                         IF #password <> #EMPTY_WSTRING AND #username <> #EMPTY_WSTRING
                         THEN
                           #tempPasswordFlag := TRUE;
                           FOR #tempLoopCounter := #FIRST_CHARACTER TO LEN(#password) DO
                             "LMQTT_ConvertToUtf8"(character     := #password[#tempLoopCounter],
                                                   convertedUtf8 => #tempConvertedUtf8,
                                                   bytesUsed     => #tempBytesUsedUtf8,
                                                   error         => #tempErrorConvertUtf8,
                                                   status        => #tempStatusConvertUtf8);
                             #statPasswordLenUtf8Encoded := #statPasswordLenUtf8Encoded + #tempBytesUsedUtf8;
                           END_FOR;
                           #statSendPaketTotalRemLen := #statSendPaketTotalRemLen + #statPasswordLenUtf8Encoded + #TWO_BYTE_LEN_INFO;
                         ELSE
                           #statPasswordEncodeState := #NOT_USED_NO_ENCODING;
                           #tempPasswordFlag := FALSE;
                         END_IF;


                         IF #willtopic <> #EMPTY_WSTRING
                         THEN
                           #tempWillFlag := TRUE;
                           CASE #statWillQos OF
                             #MQTT_QOS_0:  // Statement section case 1
                               #tempWillQoS1 := FALSE;
                               #tempWillQoS2 := FALSE;
                             #MQTT_QOS_1:  // Statement section case 2 to 4
                               #tempWillQoS1 := TRUE;
                               #tempWillQoS2 := FALSE;
                             #MQTT_QOS_2:
                               #tempWillQoS1 := FALSE;
                               #tempWillQoS2 := True;
                             ELSE  // Statement section ELSE
                               ;
                           END_CASE;
                           FOR #tempLoopCounter := #FIRST_CHARACTER TO LEN(#willtopic) DO
                             // Statement section FOR
                             "LMQTT_ConvertToUtf8"(character     := #willtopic[#tempLoopCounter],
                                                   convertedUtf8 => #tempConvertedUtf8,
                                                   bytesUsed     => #tempBytesUsedUtf8,
                                                   error         => #tempErrorConvertUtf8,
                                                   status        => #tempStatusConvertUtf8);
                             #statWillTopicLenUtf8Encoded := #statWillTopicLenUtf8Encoded + #tempBytesUsedUtf8;
                           END_FOR;
                           //Add WillTopic Len and Will Message Len (and len info twice)
                           #statSendPaketTotalRemLen := #statSendPaketTotalRemLen + #statWillTopicLenUtf8Encoded + #statWillMessageCnt + (2 * #TWO_BYTE_LEN_INFO);
                         ELSE
                           #statWillTopicEncodeState := #NOT_USED_NO_ENCODING;
                           #statWillMessageEncodeState := #NOT_USED_NO_ENCODING;
                           #tempWillFlag := FALSE;
                           #statWillRetain := FALSE;
                           #tempWillQoS1 := FALSE;
                           #tempWillQoS2 := FALSE;
                         END_IF;

                         //Build Connect Telegram
                         //Fixed Header - Write Paket Type
                         #statSendBuffer[#statSendBufferPos] := #MQTT_MSG_TYPE_CONNECT; // 1 Byte
                         #statSendBufferPos += 1; // increment

                         //Write Remaining Paket Len info 
                         WHILE (#statSendPaketTotalRemLen > #DEFAULT_VALUE_ZERO)
                         DO//See MQTT Spec for explanation of this calculation
                           #statEncodedRemPaketLenAsByte := UDINT_TO_BYTE(#statSendPaketTotalRemLen MOD #SEND_LEN_MULTIPLIER_UDINT_128);
                           #statSendPaketTotalRemLen := #statSendPaketTotalRemLen / #SEND_LEN_MULTIPLIER_UDINT_128;
                           // if there are more data to encode, set the top bit of this byte
                           IF #statSendPaketTotalRemLen > #DEFAULT_VALUE_ZERO
                           THEN
                             // Do this and continue while loop
                             #statEncodedRemPaketLenAsByte := #statEncodedRemPaketLenAsByte OR UDINT_TO_BYTE(#SEND_LEN_MULTIPLIER_UDINT_128);
                             #statSendBuffer[#statSendBufferPos] := #statEncodedRemPaketLenAsByte;
                             #statSendBufferPos += 1;
                           ELSE
                             //do this and leave while loop
                             #statSendBuffer[#statSendBufferPos] := #statEncodedRemPaketLenAsByte;
                             #statSendBufferPos += 1;
                           END_IF;
                         END_WHILE;

                         //Build Connect Telegram
                         // Write Protocol name
                         #statSendBuffer[#statSendBufferPos] := #CONN_PROTOCOL_NAME_0;
                         #statSendBufferPos += 1;
                         #statSendBuffer[#statSendBufferPos] := #CONN_PROTOCOL_NAME_4;
                         #statSendBufferPos += 1;
                         #statSendBuffer[#statSendBufferPos] := CHAR_TO_BYTE('M');
                         #statSendBufferPos += 1;
                         #statSendBuffer[#statSendBufferPos] := CHAR_TO_BYTE('Q');
                         #statSendBufferPos += 1;
                         #statSendBuffer[#statSendBufferPos] := CHAR_TO_BYTE('T');
                         #statSendBufferPos += 1;
                         #statSendBuffer[#statSendBufferPos] := CHAR_TO_BYTE('T');
                         #statSendBufferPos += 1;
                         //Write Protocol Level
                         #statSendBuffer[#statSendBufferPos] := #CONN_PROTOCOL_MQTT_VERSION_3_1_1;
                         #statSendBufferPos += 1;
                         //Write Connect Flags
                         #statSendBuffer[#statSendBufferPos].%X0 := false;
                         #statSendBuffer[#statSendBufferPos].%X1 := True;
                         #statSendBuffer[#statSendBufferPos].%X2 := #tempWillFlag;
                         #statSendBuffer[#statSendBufferPos].%X3 := #tempWillQoS1;
                         #statSendBuffer[#statSendBufferPos].%X4 := #tempWillQoS2;
                         #statSendBuffer[#statSendBufferPos].%X5 := #statWillRetain;
                         #statSendBuffer[#statSendBufferPos].%X6 := #tempPasswordFlag;
                         #statSendBuffer[#statSendBufferPos].%X7 := #tempUserFlag;
                         #statSendBufferPos += 1;
                         //Write Keep Alive in sec
                         #tempWordForSliceAddress := UINT_TO_WORD(#connParam.keepAlive);
                         #statSendBuffer[#statSendBufferPos] := #tempWordForSliceAddress.%B1;
                         #statSendBufferPos += 1;
                         #statSendBuffer[#statSendBufferPos] := #tempWordForSliceAddress.%B0;
                         #statSendBufferPos += 1;

                         //Set To Complete this, can skip in further progess
                         #statPaketHeaderEncodeDone := TRUE;
                       END_IF;

                       // Payload
                       // These fields, if present, MUST appear in the order:
                       // Client Identifier, Will topic, Will message, User Name, password


                       //ClientIdentifier
                       IF #statSendBufferPos <= #MAX_BUFFER_LEN_SEND - #TWO_BYTE_LEN_INFO THEN
                         CASE #statClientIdEncodeState OF
                           #FIRST_ENCODING:  // Statement section case 1
                             //ADD len info into paket

                             #tempWordForSliceAddress := UINT_TO_WORD(#statClientIdLenUtf8Encoded);
                             #statSendBuffer[#statSendBufferPos] := #tempWordForSliceAddress.%B1; //MSB
                             #statSendBufferPos += 1;
                             #statSendBuffer[#statSendBufferPos] := #tempWordForSliceAddress.%B0; // LSB
                             #statSendBufferPos += 1;

                             FOR #tempLoopCounter := #statClientIdPos TO LEN(#clientIdentifier) DO
                               "LMQTT_ConvertToUtf8"(character     := #clientIdentifier[#tempLoopCounter],
                                                     convertedUtf8 => #tempConvertedUtf8,
                                                     bytesUsed     => #tempBytesUsedUtf8,
                                                     error         => #tempErrorConvertUtf8,
                                                     status        => #tempStatusConvertUtf8);

                               IF #statSendBufferPos + #tempBytesUsedUtf8 <= #MAX_BUFFER_LEN_SEND THEN
                                 #statClientIdPos += 1;
                                 CASE #tempBytesUsedUtf8 OF
                                   #UTF_1_BYTE_USED:  // Statement section case 1
                                     #statSendBuffer[#statSendBufferPos] := #tempConvertedUtf8.%B0;
                                     #statSendBufferPos += 1;
                                   #UTF_2_BYTE_USED:
                                     #statSendBuffer[#statSendBufferPos] := #tempConvertedUtf8.%B0;
                                     #statSendBufferPos += 1;
                                     #statSendBuffer[#statSendBufferPos] := #tempConvertedUtf8.%B1;
                                     #statSendBufferPos += 1;
                                   #UTF_3_BYTE_USED:  // Statement section case 2 to 4
                                     #statSendBuffer[#statSendBufferPos] := #tempConvertedUtf8.%B0;
                                     #statSendBufferPos += 1;
                                     #statSendBuffer[#statSendBufferPos] := #tempConvertedUtf8.%B1;
                                     #statSendBufferPos += 1;
                                     #statSendBuffer[#statSendBufferPos] := #tempConvertedUtf8.%B2;
                                     #statSendBufferPos += 1;
                                   ELSE  // Statement section ELSE
                                     ;
                                 END_CASE;
                               ELSE
                                 //When buffer full
                                 #statClientIdEncodeState := #SUBSEQUENT_ENCODING;
                                 EXIT;
                               END_IF;
                             END_FOR;
                             IF #statClientIdPos >= LEN(#clientIdentifier) THEN
                               #statClientIdEncodeState := #ENCODE_DONE;
                             END_IF;


                           #SUBSEQUENT_ENCODING:  // Statement section case 2 to 4
                             FOR #tempLoopCounter := #statClientIdPos TO LEN(#clientIdentifier) DO
                               "LMQTT_ConvertToUtf8"(character     := #clientIdentifier[#tempLoopCounter],
                                                     convertedUtf8 => #tempConvertedUtf8,
                                                     bytesUsed     => #tempBytesUsedUtf8,
                                                     error         => #tempErrorConvertUtf8,
                                                     status        => #tempStatusConvertUtf8);
                               IF #statSendBufferPos + #tempBytesUsedUtf8 <= #MAX_BUFFER_LEN_SEND THEN
                                 #statClientIdPos += 1;
                                 CASE #tempBytesUsedUtf8 OF
                                   #UTF_1_BYTE_USED:  // Statement section case 1
                                     #statSendBuffer[#statSendBufferPos] := #tempConvertedUtf8.%B0;
                                     #statSendBufferPos += 1;
                                   #UTF_2_BYTE_USED:
                                     #statSendBuffer[#statSendBufferPos] := #tempConvertedUtf8.%B0;
                                     #statSendBufferPos += 1;
                                     #statSendBuffer[#statSendBufferPos] := #tempConvertedUtf8.%B1;
                                     #statSendBufferPos += 1;
                                   #UTF_3_BYTE_USED:  // Statement section case 2 to 4
                                     #statSendBuffer[#statSendBufferPos] := #tempConvertedUtf8.%B0;
                                     #statSendBufferPos += 1;
                                     #statSendBuffer[#statSendBufferPos] := #tempConvertedUtf8.%B1;
                                     #statSendBufferPos += 1;
                                     #statSendBuffer[#statSendBufferPos] := #tempConvertedUtf8.%B2;
                                     #statSendBufferPos += 1;
                                   ELSE  // Statement section ELSE
                                     ;
                                 END_CASE;
                               ELSE
                                 //When buffer full
                                 EXIT;
                               END_IF;
                             END_FOR;
                             IF #statClientIdPos >= LEN(#clientIdentifier) THEN
                               #statClientIdEncodeState := #ENCODE_DONE;
                             END_IF;
                           ELSE  // Statement section ELSE
                             ; // IDLE / SKIP
                         END_CASE;
                       END_IF;

                       // Will Topic
                       // If the Will Flag is set to 1, the Will Topic is the next field in the payload. It must be > 0 Bytes

                       IF #statClientIdEncodeState = #ENCODE_DONE
                         AND #statSendBufferPos <= #MAX_BUFFER_LEN_SEND - #TWO_BYTE_LEN_INFO THEN
                         //When Client Id is encoded and buffer not full
                         //And willTopic is used
                         CASE #statWillTopicEncodeState OF
                           #FIRST_ENCODING:  // Statement section case 1
                             //ADD len info into paket

                             #tempWordForSliceAddress := UINT_TO_WORD(#statWillTopicLenUtf8Encoded);
                             #statSendBuffer[#statSendBufferPos] := #tempWordForSliceAddress.%B1; //MSB
                             #statSendBufferPos += 1;
                             #statSendBuffer[#statSendBufferPos] := #tempWordForSliceAddress.%B0; // LSB
                             #statSendBufferPos += 1;

                             FOR #tempLoopCounter := #statWillTopicPos TO LEN(#willtopic) DO
                               "LMQTT_ConvertToUtf8"(character     := #willtopic[#tempLoopCounter],
                                                     convertedUtf8 => #tempConvertedUtf8,
                                                     bytesUsed     => #tempBytesUsedUtf8,
                                                     error         => #tempErrorConvertUtf8,
                                                     status        => #tempStatusConvertUtf8);

                               IF #statSendBufferPos + #tempBytesUsedUtf8 <= #MAX_BUFFER_LEN_SEND THEN
                                 //Increment when successful
                                 #statWillTopicPos += 1;

                                 CASE #tempBytesUsedUtf8 OF
                                   #UTF_1_BYTE_USED:  // Statement section case 1
                                     #statSendBuffer[#statSendBufferPos] := #tempConvertedUtf8.%B0;
                                     #statSendBufferPos += 1;
                                   #UTF_2_BYTE_USED:
                                     #statSendBuffer[#statSendBufferPos] := #tempConvertedUtf8.%B0;
                                     #statSendBufferPos += 1;
                                     #statSendBuffer[#statSendBufferPos] := #tempConvertedUtf8.%B1;
                                     #statSendBufferPos += 1;
                                   #UTF_3_BYTE_USED:  // Statement section case 2 to 4
                                     #statSendBuffer[#statSendBufferPos] := #tempConvertedUtf8.%B0;
                                     #statSendBufferPos += 1;
                                     #statSendBuffer[#statSendBufferPos] := #tempConvertedUtf8.%B1;
                                     #statSendBufferPos += 1;
                                     #statSendBuffer[#statSendBufferPos] := #tempConvertedUtf8.%B2;
                                     #statSendBufferPos += 1;
                                   ELSE  // Statement section ELSE
                                     ;
                                 END_CASE;
                               ELSE
                                 //When buffer full
                                 #statWillTopicEncodeState := #SUBSEQUENT_ENCODING;
                                 EXIT;
                               END_IF;
                             END_FOR;

                             IF #statWillTopicPos >= LEN(#willtopic) THEN
                               #statWillTopicEncodeState := #ENCODE_DONE;
                             END_IF;

                           #SUBSEQUENT_ENCODING:  // Statement section case 2 to 4
                             FOR #tempLoopCounter := #statWillTopicPos TO LEN(#willtopic) DO
                               "LMQTT_ConvertToUtf8"(character     := #willtopic[#tempLoopCounter],
                                                     convertedUtf8 => #tempConvertedUtf8,
                                                     bytesUsed     => #tempBytesUsedUtf8,
                                                     error         => #tempErrorConvertUtf8,
                                                     status        => #tempStatusConvertUtf8);

                               IF #statSendBufferPos + #tempBytesUsedUtf8 <= #MAX_BUFFER_LEN_SEND THEN
                                 #statWillTopicPos += 1;
                                 CASE #tempBytesUsedUtf8 OF
                                   #UTF_1_BYTE_USED:  // Statement section case 1
                                     #statSendBuffer[#statSendBufferPos] := #tempConvertedUtf8.%B0;
                                     #statSendBufferPos += 1;
                                   #UTF_2_BYTE_USED:
                                     #statSendBuffer[#statSendBufferPos] := #tempConvertedUtf8.%B0;
                                     #statSendBufferPos += 1;
                                     #statSendBuffer[#statSendBufferPos] := #tempConvertedUtf8.%B1;
                                     #statSendBufferPos += 1;
                                   #UTF_3_BYTE_USED:  // Statement section case 2 to 4
                                     #statSendBuffer[#statSendBufferPos] := #tempConvertedUtf8.%B0;
                                     #statSendBufferPos += 1;
                                     #statSendBuffer[#statSendBufferPos] := #tempConvertedUtf8.%B1;
                                     #statSendBufferPos += 1;
                                     #statSendBuffer[#statSendBufferPos] := #tempConvertedUtf8.%B2;
                                     #statSendBufferPos += 1;
                                   ELSE  // Statement section ELSE
                                     ;
                                 END_CASE;
                               ELSE
                                 //When buffer full
                                 EXIT;
                               END_IF;
                             END_FOR;
                             IF #statWillTopicPos >= LEN(#willtopic) THEN
                               #statWillTopicEncodeState := #ENCODE_DONE;
                             END_IF;

                           ELSE  // Statement section ELSE
                             ;
                         END_CASE;
                       END_IF;

                       // Will Message
                       // This field consists OF a two Byte length followed BY the payload FOR the Will message expressed as a sequence bytes.

                       IF #statClientIdEncodeState = #ENCODE_DONE
                         AND #statWillTopicEncodeState = #ENCODE_DONE
                         AND #statSendBufferPos <= #MAX_BUFFER_LEN_SEND - #TWO_BYTE_LEN_INFO THEN
                         //When Client Id is encoded and buffer not full
                         CASE #statWillMessageEncodeState OF
                           #FIRST_ENCODING:  // Statement section case 1
                             //ADD len info into paket

                             #tempWordForSliceAddress := UINT_TO_WORD(#statWillMessageCnt);
                             #statSendBuffer[#statSendBufferPos] := #tempWordForSliceAddress.%B1; //MSB
                             #statSendBufferPos += 1;
                             #statSendBuffer[#statSendBufferPos] := #tempWordForSliceAddress.%B0; // LSB
                             #statSendBufferPos += 1;

                             #tempLowerWillMsgArrayBoundary := LOWER_BOUND(ARR := #willMsgPayload, DIM := #ONE_DIMENSION);

                             FOR #tempLoopCounter := #statWillMessagePos TO UINT_TO_DINT(#statWillMessageCnt - 1) DO
                               IF #statSendBufferPos <= #MAX_BUFFER_LEN_SEND THEN
                                 #statSendBuffer[#statSendBufferPos] := #willMsgPayload[#tempLowerWillMsgArrayBoundary + #tempLoopCounter];
                                 #statSendBufferPos += 1;
                                 //Increment when successful
                                 #statWillMessagePos += 1;
                               ELSE
                                 //When buffer full
                                 #statWillMessageEncodeState := #SUBSEQUENT_ENCODING;
                                 EXIT;
                               END_IF;
                             END_FOR;
                             // If everything was copied successfull
                             IF #statWillMessagePos >= #statWillMessageCnt THEN
                               #statWillMessageEncodeState := #ENCODE_DONE;
                             END_IF;

                           #SUBSEQUENT_ENCODING:  // Statement section case 2 to 4
                             #tempLowerWillMsgArrayBoundary := LOWER_BOUND(ARR := #willMsgPayload, DIM := #ONE_DIMENSION);

                             FOR #tempLoopCounter := #statWillMessagePos TO UINT_TO_DINT(#statWillMessageCnt - 1) DO
                               IF #statSendBufferPos <= #MAX_BUFFER_LEN_SEND THEN
                                 #statSendBuffer[#statSendBufferPos] := #willMsgPayload[#tempLowerWillMsgArrayBoundary + #tempLoopCounter];
                                 #statSendBufferPos += 1;
                                 //Increment when successful
                                 #statWillMessagePos += 1;
                               ELSE
                                 //When Buffer Full
                                 EXIT;
                               END_IF;
                             END_FOR;
                             // If everything was copied successfull
                             IF #statWillMessagePos >= #statWillMessageCnt THEN
                               #statWillMessageEncodeState := #ENCODE_DONE;
                             END_IF;


                           ELSE  // Statement section ELSE
                             ;
                         END_CASE;
                       END_IF;

                       // Username
                       // If the Username Flag is set to 1, the Username the next field in the payload. It must be > 0 Bytes

                       IF #statClientIdEncodeState = #ENCODE_DONE
                         AND (#statWillTopicEncodeState = #ENCODE_DONE OR #statWillTopicEncodeState = #NOT_USED_NO_ENCODING)
                         AND (#statWillMessageEncodeState = #ENCODE_DONE OR #statWillTopicEncodeState = #NOT_USED_NO_ENCODING)
                         AND #statSendBufferPos <= #MAX_BUFFER_LEN_SEND - #TWO_BYTE_LEN_INFO THEN
                         //When Will Topic and Will Message is encoded and buffer not full
                         CASE #statUserNameEncodeState OF
                           #FIRST_ENCODING:  // Statement section case 1
                             //ADD len info into paket

                             #tempWordForSliceAddress := UINT_TO_WORD(#statUsernameLenUtf8Encoded);
                             #statSendBuffer[#statSendBufferPos] := #tempWordForSliceAddress.%B1; //MSB
                             #statSendBufferPos += 1;
                             #statSendBuffer[#statSendBufferPos] := #tempWordForSliceAddress.%B0; // LSB
                             #statSendBufferPos += 1;

                             FOR #tempLoopCounter := #statUserNamePos TO LEN(#username) DO
                               "LMQTT_ConvertToUtf8"(character     := #username[#tempLoopCounter],
                                                     convertedUtf8 => #tempConvertedUtf8,
                                                     bytesUsed     => #tempBytesUsedUtf8,
                                                     error         => #tempErrorConvertUtf8,
                                                     status        => #tempStatusConvertUtf8);

                               IF #statSendBufferPos + #tempBytesUsedUtf8 <= #MAX_BUFFER_LEN_SEND THEN
                                 //Increment when successful
                                 #statUserNamePos += 1;

                                 CASE #tempBytesUsedUtf8 OF
                                   #UTF_1_BYTE_USED:  // Statement section case 1
                                     #statSendBuffer[#statSendBufferPos] := #tempConvertedUtf8.%B0;
                                     #statSendBufferPos += 1;
                                   #UTF_2_BYTE_USED:
                                     #statSendBuffer[#statSendBufferPos] := #tempConvertedUtf8.%B0;
                                     #statSendBufferPos += 1;
                                     #statSendBuffer[#statSendBufferPos] := #tempConvertedUtf8.%B1;
                                     #statSendBufferPos += 1;
                                   #UTF_3_BYTE_USED:  // Statement section case 2 to 4
                                     #statSendBuffer[#statSendBufferPos] := #tempConvertedUtf8.%B0;
                                     #statSendBufferPos += 1;
                                     #statSendBuffer[#statSendBufferPos] := #tempConvertedUtf8.%B1;
                                     #statSendBufferPos += 1;
                                     #statSendBuffer[#statSendBufferPos] := #tempConvertedUtf8.%B2;
                                     #statSendBufferPos += 1;
                                   ELSE  // Statement section ELSE
                                     ;
                                 END_CASE;
                               ELSE
                                 //When buffer full
                                 #statUserNameEncodeState := #SUBSEQUENT_ENCODING;
                                 EXIT;
                               END_IF;
                             END_FOR;

                             IF #statUserNamePos >= LEN(#username) THEN
                               #statUserNameEncodeState := #ENCODE_DONE;
                             END_IF;

                           #SUBSEQUENT_ENCODING:  // Statement section case 2 to 4
                             FOR #tempLoopCounter := #statUserNamePos TO LEN(#username) DO
                               "LMQTT_ConvertToUtf8"(character     := #username[#tempLoopCounter],
                                                     convertedUtf8 => #tempConvertedUtf8,
                                                     bytesUsed     => #tempBytesUsedUtf8,
                                                     error         => #tempErrorConvertUtf8,
                                                     status        => #tempStatusConvertUtf8);

                               IF #statSendBufferPos + #tempBytesUsedUtf8 <= #MAX_BUFFER_LEN_SEND THEN
                                 #statUserNamePos += 1;
                                 CASE #tempBytesUsedUtf8 OF
                                   #UTF_1_BYTE_USED:  // Statement section case 1
                                     #statSendBuffer[#statSendBufferPos] := #tempConvertedUtf8.%B0;
                                     #statSendBufferPos += 1;
                                   #UTF_2_BYTE_USED:
                                     #statSendBuffer[#statSendBufferPos] := #tempConvertedUtf8.%B0;
                                     #statSendBufferPos += 1;
                                     #statSendBuffer[#statSendBufferPos] := #tempConvertedUtf8.%B1;
                                     #statSendBufferPos += 1;
                                   #UTF_3_BYTE_USED:  // Statement section case 2 to 4
                                     #statSendBuffer[#statSendBufferPos] := #tempConvertedUtf8.%B0;
                                     #statSendBufferPos += 1;
                                     #statSendBuffer[#statSendBufferPos] := #tempConvertedUtf8.%B1;
                                     #statSendBufferPos += 1;
                                     #statSendBuffer[#statSendBufferPos] := #tempConvertedUtf8.%B2;
                                     #statSendBufferPos += 1;
                                   ELSE  // Statement section ELSE
                                     ;
                                 END_CASE;
                               ELSE
                                 //When buffer full
                                 EXIT;
                               END_IF;
                             END_FOR;
                             IF #statUserNamePos >= LEN(#username) THEN
                               #statUserNameEncodeState := #ENCODE_DONE;
                             END_IF;

                           ELSE  // Statement section ELSE
                             ;
                         END_CASE;
                       END_IF;

                       // Password
                       // If the Password Flag is set to 1, the Password the next field in the payload. It must be > 0 Bytes
                       //Password field contains 0 to 65535 bytes OF binary data prefixed with a two Byte length field which indicates the number OF bytes used

                       IF #statClientIdEncodeState = #ENCODE_DONE
                         AND (#statWillTopicEncodeState = #ENCODE_DONE OR #statWillTopicEncodeState = #NOT_USED_NO_ENCODING)
                         AND (#statWillMessageEncodeState = #ENCODE_DONE OR #statWillMessageEncodeState = #NOT_USED_NO_ENCODING)
                         AND (#statUserNameEncodeState = #ENCODE_DONE OR #statUserNameEncodeState = #NOT_USED_NO_ENCODING)
                         AND #statSendBufferPos <= #MAX_BUFFER_LEN_SEND - #TWO_BYTE_LEN_INFO THEN
                         //When Will Topic and Will Message is encoded and buffer not full
                         CASE #statPasswordEncodeState OF
                           #FIRST_ENCODING:  // Statement section case 1
                             //ADD len info into paket

                             #tempWordForSliceAddress := UINT_TO_WORD(#statPasswordLenUtf8Encoded);
                             #statSendBuffer[#statSendBufferPos] := #tempWordForSliceAddress.%B1; //MSB
                             #statSendBufferPos += 1;
                             #statSendBuffer[#statSendBufferPos] := #tempWordForSliceAddress.%B0; // LSB
                             #statSendBufferPos += 1;

                             FOR #tempLoopCounter := #statPasswordPos TO LEN(#password) DO
                               "LMQTT_ConvertToUtf8"(character     := #password[#tempLoopCounter],
                                                     convertedUtf8 => #tempConvertedUtf8,
                                                     bytesUsed     => #tempBytesUsedUtf8,
                                                     error         => #tempErrorConvertUtf8,
                                                     status        => #tempStatusConvertUtf8);

                               IF #statSendBufferPos + #tempBytesUsedUtf8 <= #MAX_BUFFER_LEN_SEND THEN
                                 //Increment when successful
                                 #statPasswordPos += 1;

                                 CASE #tempBytesUsedUtf8 OF
                                   #UTF_1_BYTE_USED:  // Statement section case 1
                                     #statSendBuffer[#statSendBufferPos] := #tempConvertedUtf8.%B0;
                                     #statSendBufferPos += 1;
                                   #UTF_2_BYTE_USED:
                                     #statSendBuffer[#statSendBufferPos] := #tempConvertedUtf8.%B0;
                                     #statSendBufferPos += 1;
                                     #statSendBuffer[#statSendBufferPos] := #tempConvertedUtf8.%B1;
                                     #statSendBufferPos += 1;
                                   #UTF_3_BYTE_USED:  // Statement section case 2 to 4
                                     #statSendBuffer[#statSendBufferPos] := #tempConvertedUtf8.%B0;
                                     #statSendBufferPos += 1;
                                     #statSendBuffer[#statSendBufferPos] := #tempConvertedUtf8.%B1;
                                     #statSendBufferPos += 1;
                                     #statSendBuffer[#statSendBufferPos] := #tempConvertedUtf8.%B2;
                                     #statSendBufferPos += 1;
                                   ELSE  // Statement section ELSE
                                     ;
                                 END_CASE;
                               ELSE
                                 //When buffer full
                                 #statPasswordEncodeState := #SUBSEQUENT_ENCODING;
                                 EXIT;
                               END_IF;
                             END_FOR;

                             IF #statPasswordPos >= LEN(#password) THEN
                               #statPasswordEncodeState := #ENCODE_DONE;
                             END_IF;

                           #SUBSEQUENT_ENCODING:  // Statement section case 2 to 4
                             FOR #tempLoopCounter := #statPasswordPos TO LEN(#password) DO
                               "LMQTT_ConvertToUtf8"(character     := #password[#tempLoopCounter],
                                                     convertedUtf8 => #tempConvertedUtf8,
                                                     bytesUsed     => #tempBytesUsedUtf8,
                                                     error         => #tempErrorConvertUtf8,
                                                     status        => #tempStatusConvertUtf8);

                               IF #statSendBufferPos + #tempBytesUsedUtf8 <= #MAX_BUFFER_LEN_SEND THEN
                                 #statPasswordPos += 1;
                                 CASE #tempBytesUsedUtf8 OF
                                   #UTF_1_BYTE_USED:  // Statement section case 1
                                     #statSendBuffer[#statSendBufferPos] := #tempConvertedUtf8.%B0;
                                     #statSendBufferPos += 1;
                                   #UTF_2_BYTE_USED:
                                     #statSendBuffer[#statSendBufferPos] := #tempConvertedUtf8.%B0;
                                     #statSendBufferPos += 1;
                                     #statSendBuffer[#statSendBufferPos] := #tempConvertedUtf8.%B1;
                                     #statSendBufferPos += 1;
                                   #UTF_3_BYTE_USED:  // Statement section case 2 to 4
                                     #statSendBuffer[#statSendBufferPos] := #tempConvertedUtf8.%B0;
                                     #statSendBufferPos += 1;
                                     #statSendBuffer[#statSendBufferPos] := #tempConvertedUtf8.%B1;
                                     #statSendBufferPos += 1;
                                     #statSendBuffer[#statSendBufferPos] := #tempConvertedUtf8.%B2;
                                     #statSendBufferPos += 1;
                                   ELSE  // Statement section ELSE
                                     ;
                                 END_CASE;
                               ELSE
                                 //When buffer full
                                 EXIT;
                               END_IF;
                             END_FOR;
                             IF #statPasswordPos >= LEN(#password) THEN
                               #statPasswordEncodeState := #ENCODE_DONE;
                             END_IF;

                           ELSE  // Statement section ELSE
                             ;
                         END_CASE;
                       END_IF;

                       //set Sendlen for TSendC Block

                       #statTsendcLen := #statSendBufferPos; // Buffer pos equals amount of elements in send array
                       //reset buffer pos
                       #statSendBufferPos := 0;
                       //enable Send Req
                       #statTsendcReq := TRUE;
                       //Set Watchdog
                       #statEnableTimerCommandWatchdog := TRUE;
                       //wait for send to be done
                       #statMqttConnectState := #MQTT_CONNECT_STATE_SEND_PAKET_WAIT_FOR_CONNACK;
                     END_IF;
                   END_REGION BUILD_CONNECT_PAKET
                 #MQTT_CONNECT_STATE_SEND_PAKET_WAIT_FOR_CONNACK:
                   REGION SEND_CONNECT_PAKET_WAIT_FOR_CONNACK
                     //check tsend status
                     IF NOT #tempTsendcBusy AND #tempTsendcStatus = #TSENDC_JOB_DONE THEN
                       IF (#statClientIdEncodeState = #ENCODE_DONE OR #statClientIdEncodeState = #NOT_USED_NO_ENCODING)
                         AND (#statWillTopicEncodeState = #ENCODE_DONE OR #statWillTopicEncodeState = #NOT_USED_NO_ENCODING)
                         AND (#statWillMessageEncodeState = #ENCODE_DONE OR #statWillMessageEncodeState = #NOT_USED_NO_ENCODING)
                         AND (#statUserNameEncodeState = #ENCODE_DONE OR #statUserNameEncodeState = #NOT_USED_NO_ENCODING)
                         AND (#statPasswordEncodeState = #ENCODE_DONE OR #statPasswordEncodeState = #NOT_USED_NO_ENCODING) THEN
                         //Encoding done all sent
                         #statPaketHeaderEncodeDone := FALSE;
                       ELSE
                         // More to Encode and send
                         #statEnableTimerCommandWatchdog := FALSE;
                         #statMqttConnectState := #MQTT_CONNECT_STATE_BUILD_PAKET;
                       END_IF;
                     END_IF;
                     //Check watchdog
                     IF #instTimerCommandWatchdog.Q THEN
                       #statEnableTimerCommandWatchdog := FALSE;
                       #statPaketHeaderEncodeDone := FALSE;
                       #statStatus := #ERR_MQTT_CONNECT_TIMEOUT; // Set correct status that identifies error clearly
                       #statSubfunctionStatus := #ERR_MQTT_CONNECT_TIMEOUT; // Status or return value of called FBs, FCs and system blocks
                       #statFBErrorState := #statFBState; // Set error state number for diagnostic 
                       #statErrorAutoCleared := TRUE;
                       #statMqttConnectState := #MQTT_CONNECT_STATE_BUILD_PAKET;
                     END_IF;

                     //Check Connect ACK paket
                     CASE #tempMqttConnAckRcvStatus OF
                       #NO_RESPONSE:  //  IDLE
                         ;
                       #RESPONSE_GOOD:  // Statement section case 2 to 4
                         //disable watchdog
                         #statEnableTimerCommandWatchdog := FALSE;
                         //Encoding done all sent
                         #statPaketHeaderEncodeDone := FALSE;
                         //Go to Connected
                         #statMqttConnectState := #MQTT_CONNECT_STATE_CONNECTED;
                         #statStatus := #STATUS_MQTT_CONNECTED;
                     END_CASE;
                   END_REGION REGION SEND_CONNECT_PAKET
                 #MQTT_CONNECT_STATE_CONNECTED:
                   REGION CONNECTED
                     //Check Rising edge of input commands
                     #tempCommandInput.%X0 := #tempPublish AND NOT #statPublishOld;
                     #tempCommandInput.%X1 := #tempSubscribe AND NOT #statSubscribeOld;
                     #tempCommandInput.%X2 := #tempUnsubscribe AND NOT #statUnsubscribeOld;

                     //Start the keepalive timer if used
                     #statEnableMqttKeepAliveTimer := #statMqttKeepAliveUsed;

                     //set status to connected after successfully executed job
                     IF #statStatus = #STATUS_JOB_EXECUTED THEN
                       #statStatus := #STATUS_MQTT_CONNECTED;
                     END_IF;

                     REGION MQTT_COMMANDS
                       //When state machine is ready for a new input then assign correct command
                       //Ping job can be overwritten by a command.
                         IF #tempCommandInput <> #NO_COMMAND
                         AND (#statMqttCommandState = #MQTT_COMMAND_STATE_NO_PROCESSING OR #statMqttCommandState = #MQTT_COMMAND_STATE_SEND_PING)
                       THEN
                         // New Input set, reset done flag
                         #statDone := FALSE;
                         #statMqttCommandState := BYTE_TO_DINT(#tempCommandInput);
                       END_IF;

                       CASE #statMqttCommandState OF
                         #MQTT_COMMAND_STATE_NO_PROCESSING:
                           //EMPTY STATE
                           ;
                         #MQTT_COMMAND_STATE_BUILD_PUBLISH:  // Statement section case 1
                           REGION PUBLISH_TO_TOPIC
                             //Remaining Length is the length of the variable header (TOPIC NAME + PacketID) plus the length of the Payload. 
                             //Max Len of Mqtt pakets is per Standard 268,435,455 Bytes (ff,ff,ff,7f)
                             //Calculate Remain Len will be
                             //Len of TOPIC   (max 3*16382 WChars= 49.146 Bytes)
                             //plus Len of PacketID (2 Bytes)
                             //plus Len of Payload (max 268,435,455 - 49.146 - 2 = 268.386.307 Bytes ca. 268 MB)
                             //Max Array / DB Len in TIA portal is around 16 MB or 16.777.216 Byte
                             //Set Status
                             #statStatus := #STATUS_MQTT_PUBLISH;

                             // Must obey, if not currently sending PubAck Msg on a subscription
                             // Else, try in the next cycle
                             IF #tempTsendcBusy = FALSE // when tsendC is ready
                               AND #tempTsendcDone = FALSE // tsendC did not finish in this cycle
                               AND #statTsendcReq = FALSE // TsendC request was not already requested by pub ack msg
                             THEN
                               IF #statPaketHeaderEncodeDone = FALSE THEN

                                 //Init
                                 #statSendPaketTotalRemLen := 0;
                                 #statSendBufferPos := 0;
                                 #statPublishQos := #qos;
                                 #statPublishMessageCnt := #publishMsgLen;
                                 #statPublishTopicEncodeState := #FIRST_ENCODING;
                                 #statPublishTopicPos := #FIRST_CHARACTER;
                                 #statPublishTopicLenUtf8Encoded := 0;
                                 #statPaketId += 1;//increment
                                 #statPaketIdEncoded := FALSE;
                                 #statPublishEncodeMessageState := #SUBSEQUENT_ENCODING; // No len info necessary so start directly at subsequent.
                                 #statPublishMessagePos := 0; // first array element

                                 //verify PayloadLen
                                 #tempMaxPublishDataArrayLen := ABS(UPPER_BOUND(ARR := #publishMsgPayload, DIM := #ONE_DIMENSION) - LOWER_BOUND(ARR := #publishMsgPayload, DIM := #ONE_DIMENSION)) + #ARRAY_LEN_OFFSET_PLUS_1;

                                 //check necessary boundaries
                                 IF #tempMaxPublishDataArrayLen < #statPublishMessageCnt THEN
                                   #statStatus := #ERR_CNT_EXCEEDS_ARRAY_DIMENSION; // Set correct status that identifies error clearly
                                   #statSubfunctionStatus := #ERR_CNT_EXCEEDS_ARRAY_DIMENSION; // Status or return value of called FBs, FCs and system blocks
                                   #statFBErrorState := #statFBState; // Set error state number for diagnostic 
                                   #statErrorAutoCleared := TRUE;
                                   #statMqttCommandState := #MQTT_COMMAND_STATE_NO_PROCESSING;
                                 ELSIF LEN(#mqttTopic) = #LEN_NULL THEN
                                   #statStatus := #ERR_MQTT_COMMAND_PUBLISH_TOPIC_INVALID; // Set correct status that identifies error clearly
                                   #statSubfunctionStatus := #ERR_MQTT_COMMAND_PUBLISH_TOPIC_INVALID; // Status or return value of called FBs, FCs and system blocks
                                   #statFBErrorState := #statFBState; // Set error state number for diagnostic 
                                   #statErrorAutoCleared := TRUE;
                                   #statMqttCommandState := #MQTT_COMMAND_STATE_NO_PROCESSING;
                                 ELSIF #statPublishQos > #MQTT_QOS_2 THEN
                                   #statStatus := #ERR_QOS_INVALID; // Set correct status that identifies error clearly
                                   #statSubfunctionStatus := #ERR_QOS_INVALID; // Status or return value of called FBs, FCs and system blocks
                                   #statFBErrorState := #statFBState; // Set error state number for diagnostic 
                                   #statErrorAutoCleared := TRUE;
                                   #statMqttCommandState := #MQTT_COMMAND_STATE_NO_PROCESSING;
                                 ELSE // All ok
                                   //Add amount of bytes for publish message
                                   #statSendPaketTotalRemLen := #statSendPaketTotalRemLen + #statPublishMessageCnt;
                                   //add publish  topic len
                                   FOR #tempLoopCounter := #FIRST_CHARACTER TO LEN(#mqttTopic) DO
                                     "LMQTT_ConvertToUtf8"(character     := #mqttTopic[#tempLoopCounter],
                                                           convertedUtf8 => #tempConvertedUtf8,
                                                           bytesUsed     => #tempBytesUsedUtf8,
                                                           error         => #tempErrorConvertUtf8,
                                                           status        => #tempStatusConvertUtf8);
                                     #statPublishTopicLenUtf8Encoded := #statPublishTopicLenUtf8Encoded + #tempBytesUsedUtf8;
                                   END_FOR;
                                   #statSendPaketTotalRemLen := #statSendPaketTotalRemLen + #statPublishTopicLenUtf8Encoded + #TWO_BYTE_LEN_INFO;

                                   //Build Publish Telegram
                                   //Fixed Header - Write Paket Type
                                   #statSendBuffer[#statSendBufferPos] := #MQTT_MSG_TYPE_PUBLISH;
                                   // Set DUP flag always to FALSE
                                   #statSendBuffer[#statSendBufferPos].%X3 := FALSE;
                                   // Set QoS Level
                                   CASE #statPublishQos OF
                                     #MQTT_QOS_0:  // Statement section case 0
                                       #statSendBuffer[#statSendBufferPos].%X2 := FALSE;
                                       #statSendBuffer[#statSendBufferPos].%X1 := FALSE;
                                     #MQTT_QOS_1:  // Statement section case 1
                                       #statSendBuffer[#statSendBufferPos].%X2 := FALSE;
                                       #statSendBuffer[#statSendBufferPos].%X1 := TRUE;
                                       //Add two byte len info for Mandatory packet ID
                                       #statSendPaketTotalRemLen := #statSendPaketTotalRemLen + #TWO_BYTE_LEN_INFO;
                                     #MQTT_QOS_2: // Statement section case 2
                                       #statSendBuffer[#statSendBufferPos].%X2 := TRUE;
                                       #statSendBuffer[#statSendBufferPos].%X1 := FALSE;
                                       //Add two byte len info for Mandatory packet ID
                                       #statSendPaketTotalRemLen := #statSendPaketTotalRemLen + #TWO_BYTE_LEN_INFO;
                                     ELSE
                                       ;
                                   END_CASE;
                                   //Set retain bit
                                   #statSendBuffer[#statSendBufferPos].%X0 := #retain;

                                   #statSendBufferPos += 1; // increment

                                   //Write Remaining Paket Len info 
                                   WHILE (#statSendPaketTotalRemLen > #DEFAULT_VALUE_ZERO)
                                   DO//See MQTT Spec for explanation of this calculation
                                     #statEncodedRemPaketLenAsByte := UDINT_TO_BYTE(#statSendPaketTotalRemLen MOD #SEND_LEN_MULTIPLIER_UDINT_128);
                                     #statSendPaketTotalRemLen := #statSendPaketTotalRemLen / #SEND_LEN_MULTIPLIER_UDINT_128;
                                     // if there are more data to encode, set the top bit of this byte
                                     IF #statSendPaketTotalRemLen > #DEFAULT_VALUE_ZERO
                                     THEN
                                       // Do this and continue while loop
                                       #statEncodedRemPaketLenAsByte := #statEncodedRemPaketLenAsByte OR UDINT_TO_BYTE(#SEND_LEN_MULTIPLIER_UDINT_128);
                                       #statSendBuffer[#statSendBufferPos] := #statEncodedRemPaketLenAsByte;
                                       #statSendBufferPos += 1;
                                     ELSE
                                       //do this and leave while loop
                                       #statSendBuffer[#statSendBufferPos] := #statEncodedRemPaketLenAsByte;
                                       #statSendBufferPos += 1;
                                     END_IF;
                                   END_WHILE;
                                   //When all done, set encode to true
                                   #statPaketHeaderEncodeDone := TRUE;
                                 END_IF;
                               END_IF;

                               //Header Encoded - now Topic, PacketId and Message need to be encoded.
                               IF #statPaketHeaderEncodeDone = TRUE THEN

                                 //Publish Topic
                                 IF #statSendBufferPos <= #MAX_BUFFER_LEN_SEND - #TWO_BYTE_LEN_INFO THEN
                                   CASE #statPublishTopicEncodeState OF
                                     #FIRST_ENCODING:  // Statement section case 1
                                       //ADD len info into paket

                                       #tempWordForSliceAddress := UINT_TO_WORD(#statPublishTopicLenUtf8Encoded);
                                       #statSendBuffer[#statSendBufferPos] := #tempWordForSliceAddress.%B1; //MSB
                                       #statSendBufferPos += 1;
                                       #statSendBuffer[#statSendBufferPos] := #tempWordForSliceAddress.%B0; // LSB
                                       #statSendBufferPos += 1;

                                       FOR #tempLoopCounter := #statPublishTopicPos TO LEN(#mqttTopic) DO
                                         "LMQTT_ConvertToUtf8"(character     := #mqttTopic[#tempLoopCounter],
                                                               convertedUtf8 => #tempConvertedUtf8,
                                                               bytesUsed     => #tempBytesUsedUtf8,
                                                               error         => #tempErrorConvertUtf8,
                                                               status        => #tempStatusConvertUtf8);

                                         IF #statSendBufferPos + #tempBytesUsedUtf8 <= #MAX_BUFFER_LEN_SEND THEN
                                           #statPublishTopicPos += 1;
                                           CASE #tempBytesUsedUtf8 OF
                                             #UTF_1_BYTE_USED:  // Statement section case 1
                                               #statSendBuffer[#statSendBufferPos] := #tempConvertedUtf8.%B0;
                                               #statSendBufferPos += 1;
                                             #UTF_2_BYTE_USED:
                                               #statSendBuffer[#statSendBufferPos] := #tempConvertedUtf8.%B0;
                                               #statSendBufferPos += 1;
                                               #statSendBuffer[#statSendBufferPos] := #tempConvertedUtf8.%B1;
                                               #statSendBufferPos += 1;
                                             #UTF_3_BYTE_USED:  // Statement section case 2 to 4
                                               #statSendBuffer[#statSendBufferPos] := #tempConvertedUtf8.%B0;
                                               #statSendBufferPos += 1;
                                               #statSendBuffer[#statSendBufferPos] := #tempConvertedUtf8.%B1;
                                               #statSendBufferPos += 1;
                                               #statSendBuffer[#statSendBufferPos] := #tempConvertedUtf8.%B2;
                                               #statSendBufferPos += 1;
                                             ELSE  // Statement section ELSE
                                               ;
                                           END_CASE;
                                         ELSE
                                           //When buffer full
                                           #statPublishTopicEncodeState := #SUBSEQUENT_ENCODING;
                                           EXIT;
                                         END_IF;
                                       END_FOR;
                                       IF #statPublishTopicPos >= LEN(#mqttTopic) THEN
                                         #statPublishTopicEncodeState := #ENCODE_DONE;
                                       END_IF;


                                     #SUBSEQUENT_ENCODING:  // Statement section case 2 to 4
                                       FOR #tempLoopCounter := #statPublishTopicPos TO LEN(#mqttTopic) DO

                                         "LMQTT_ConvertToUtf8"(character     := #mqttTopic[#tempLoopCounter],
                                                               convertedUtf8 => #tempConvertedUtf8,
                                                               bytesUsed     => #tempBytesUsedUtf8,
                                                               error         => #tempErrorConvertUtf8,
                                                               status        => #tempStatusConvertUtf8);
                                         IF #statSendBufferPos + #tempBytesUsedUtf8 <= #MAX_BUFFER_LEN_SEND THEN
                                           #statPublishTopicPos += 1;
                                           CASE #tempBytesUsedUtf8 OF
                                             #UTF_1_BYTE_USED:  // Statement section case 1
                                               #statSendBuffer[#statSendBufferPos] := #tempConvertedUtf8.%B0;
                                               #statSendBufferPos += 1;
                                             #UTF_2_BYTE_USED:
                                               #statSendBuffer[#statSendBufferPos] := #tempConvertedUtf8.%B0;
                                               #statSendBufferPos += 1;
                                               #statSendBuffer[#statSendBufferPos] := #tempConvertedUtf8.%B1;
                                               #statSendBufferPos += 1;
                                             #UTF_3_BYTE_USED:  // Statement section case 2 to 4
                                               #statSendBuffer[#statSendBufferPos] := #tempConvertedUtf8.%B0;
                                               #statSendBufferPos += 1;
                                               #statSendBuffer[#statSendBufferPos] := #tempConvertedUtf8.%B1;
                                               #statSendBufferPos += 1;
                                               #statSendBuffer[#statSendBufferPos] := #tempConvertedUtf8.%B2;
                                               #statSendBufferPos += 1;
                                             ELSE  // Statement section ELSE
                                               ;
                                           END_CASE;
                                         ELSE
                                           //When buffer full
                                           EXIT;
                                         END_IF;
                                       END_FOR;
                                       IF #statPublishTopicPos >= LEN(#mqttTopic) THEN
                                         #statPublishTopicEncodeState := #ENCODE_DONE;
                                       END_IF;
                                     ELSE  // SKIP if done
                                       ;
                                   END_CASE;
                                 END_IF;

                                 // Encode MessageID, when QOS > 0 and  Topic done and buffer not full
                                 IF #statPublishTopicEncodeState = #ENCODE_DONE
                                   AND #statPaketIdEncoded = FALSE
                                   AND #statSendBufferPos <= #MAX_BUFFER_LEN_SEND - #TWO_BYTE_LEN_INFO THEN
                                   // Check QoS - only necessary if QoS >0
                                   CASE #statPublishQos OF
                                     #MQTT_QOS_1:
                                       #tempWordForSliceAddress := UINT_TO_WORD(#statPaketId);
                                       #statSendBuffer[#statSendBufferPos] := #tempWordForSliceAddress.%B1; //MSB
                                       #statSendBufferPos += 1;
                                       #statSendBuffer[#statSendBufferPos] := #tempWordForSliceAddress.%B0; //LSB
                                       #statSendBufferPos += 1;
                                     #MQTT_QOS_2:
                                       #tempWordForSliceAddress := UINT_TO_WORD(#statPaketId);
                                       #statSendBuffer[#statSendBufferPos] := #tempWordForSliceAddress.%B1; //MSB
                                       #statSendBufferPos += 1;
                                       #statSendBuffer[#statSendBufferPos] := #tempWordForSliceAddress.%B0; //LSB
                                       #statSendBufferPos += 1;
                                     ELSE
                                       //No paket id to encode here
                                       ;
                                   END_CASE;
                                   //Finally:
                                   #statPaketIdEncoded := TRUE;
                                 END_IF;

                                 // Encode Payload, when  Topic done and PaketID Done and buffer not full
                                 IF #statPublishTopicEncodeState = #ENCODE_DONE
                                   AND #statPaketIdEncoded = TRUE
                                   AND #statSendBufferPos < #MAX_BUFFER_LEN_SEND THEN

                                   // Publish Message Encoding
                                   // This Contains the payload from the publish message expressed as a sequence bytes.
                                   CASE #statPublishEncodeMessageState OF
                                     #SUBSEQUENT_ENCODING:  // Statement section case 2 to 4
                                       #tempLowerBoundPublishDataArray := LOWER_BOUND(ARR := #publishMsgPayload, DIM := #ONE_DIMENSION);

                                       FOR #tempLoopCounter := #statPublishMessagePos TO UDINT_TO_DINT(#statPublishMessageCnt - 1) DO
                                         IF #statSendBufferPos <= #MAX_BUFFER_LEN_SEND THEN
                                           #statSendBuffer[#statSendBufferPos] := #publishMsgPayload[#tempLowerBoundPublishDataArray + #tempLoopCounter];
                                           #statSendBufferPos += 1;
                                           //Increment when successful
                                           #statPublishMessagePos += 1;
                                         ELSE
                                           //When Buffer Full
                                           EXIT;
                                         END_IF;
                                       END_FOR;
                                       // If everything was copied successfull
                                       IF #statPublishMessagePos >= #statPublishMessageCnt THEN
                                         #statPublishEncodeMessageState := #ENCODE_DONE;
                                       END_IF;
                                     ELSE  // Statement section ELSE
                                       ;
                                   END_CASE;
                                 END_IF;


                                 //set Sendlen for TSendC Block
                                 #statTsendcLen := #statSendBufferPos; // Buffer pos equals amount of elements in send array
                                 //reset buffer pos
                                 #statSendBufferPos := 0;
                                 //enable Send Req
                                 #statTsendcReq := TRUE;
                                 //Set Watchdog
                                 #statEnableTimerCommandWatchdog := TRUE;
                                 //wait for send to be done
                                 #statMqttCommandState := #MQTT_COMMAND_STATE_SEND_PUBLISH;
                               END_IF;
                             END_IF;

                           END_REGION PUBLISH_TO_TOPIC
                         #MQTT_COMMAND_STATE_SEND_PUBLISH:
                           REGION SEND_PUBLISH_WAIT_FOR_RESPONSE
                             //check tsend status
                             IF NOT #tempTsendcBusy AND #tempTsendcStatus = #TSENDC_JOB_DONE THEN
                               IF (#statPublishTopicEncodeState = #ENCODE_DONE)
                                 AND (#statPublishEncodeMessageState = #ENCODE_DONE) THEN
                                 //Encoding done all sent
                                 #statPaketHeaderEncodeDone := FALSE;
                                 //  with QoS = 0 Job done
                                 IF #statPublishQos = #MQTT_QOS_0 THEN
                                   // job done
                                   #statDone := TRUE;
                                   // go back to idle
                                   #statMqttCommandState := #MQTT_COMMAND_STATE_NO_PROCESSING;
                                   //reset Watchdog
                                   #statEnableTimerCommandWatchdog := FALSE;
                                   // Set Status back to connected
                                   #statStatus := #STATUS_JOB_EXECUTED;
                                 END_IF;
                               ELSE
                                 // More to Encode and send
                                 #statEnableTimerCommandWatchdog := FALSE;
                                 #statMqttCommandState := #MQTT_COMMAND_STATE_BUILD_PUBLISH;
                               END_IF;
                             END_IF;
                             //check watchdog
                             IF #instTimerCommandWatchdog.Q THEN
                               #statEnableTimerCommandWatchdog := FALSE;
                               #statStatus := #ERR_MQTT_COMMAND_SEND_TIMEOUT; // Set correct status that identifies error clearly
                               #statSubfunctionStatus := #ERR_MQTT_COMMAND_SEND_TIMEOUT; // Status or return value of called FBs, FCs and system blocks
                               #statFBErrorState := #statFBState; // Set error state number for diagnostic 
                               #statErrorAutoCleared := TRUE;
                               #statMqttCommandState := #MQTT_COMMAND_STATE_NO_PROCESSING;
                             END_IF;

                             //When QoS = 1; Wait for Publish ACK paket
                             CASE #tempMqttPubAckRcv OF
                               #NO_RESPONSE:  // Statement section case 0 IDLE
                                 ;
                               #RESPONSE_GOOD:  // Statement section case 1 OKAY
                                 //disable watchdog
                                 #statEnableTimerCommandWatchdog := FALSE;
                                 //Encoding done all sent
                                 #statPaketHeaderEncodeDone := FALSE;
                                 //Publish QoS 1 = Done
                                 #statDone := TRUE;
                                 #statMqttCommandState := #MQTT_COMMAND_STATE_NO_PROCESSING;
                                 // Set Status back to connected
                                 #statStatus := #STATUS_JOB_EXECUTED;
                               #RESPONSE_PAKET_ID_INVALID:
                                 #statStatus := #ERR_MQTT_PAKET_ID_INVALID; // Set correct status that identifies error clearly
                                 #statSubfunctionStatus := #ERR_MQTT_PAKET_ID_INVALID; // Status or return value of called FBs, FCs and system blocks
                                 #statFBErrorState := #statFBState; // Set error state number for diagnostic 
                                 #statErrorAutoCleared := TRUE;
                                 #statMqttCommandState := #MQTT_COMMAND_STATE_NO_PROCESSING;
                             END_CASE;

                             //When QOS = 2 and Pub Rec Receieved:
                             CASE #tempMqttPubRecRcv OF
                               #NO_RESPONSE:  // 0 IDLE
                                 ;
                               #RESPONSE_GOOD:
                                 //Encoding done all sent
                                 #statPaketHeaderEncodeDone := FALSE;
                                 // Send Publish Release paket
                                 #statSendBufferPos := 0;
                                 #statSendBuffer[#statSendBufferPos] := #MQTT_MSG_TYPE_PUBREL;
                                 #statSendBufferPos += 1;
                                 //Remaining Lenght (must be 2)
                                 #statSendBuffer[#statSendBufferPos] := #REMAINING_LEN_2;
                                 #statSendBufferPos += 1;
                                 // add paket id 
                                 #tempWordForSliceAddress := UINT_TO_WORD(#statPaketId);
                                 #statSendBuffer[#statSendBufferPos] := #tempWordForSliceAddress.%B1; //MSB
                                 #statSendBufferPos += 1;
                                 #statSendBuffer[#statSendBufferPos] := #tempWordForSliceAddress.%B0; //LSB
                                 #statSendBufferPos += 1;
                                 #statTsendcLen := #statSendBufferPos;
                                 //Start send request
                                 #statTsendcReq := TRUE;
                                 //Reset watchdog and start
                                 RESET_TIMER(#instTimerCommandWatchdog);
                                 #statEnableTimerCommandWatchdog := TRUE;
                                 //Stay in State
                               #RESPONSE_PAKET_ID_INVALID:
                                 #statStatus := #ERR_MQTT_PAKET_ID_INVALID; // Set correct status that identifies error clearly
                                 #statSubfunctionStatus := #ERR_MQTT_PAKET_ID_INVALID; // Status or return value of called FBs, FCs and system blocks
                                 #statFBErrorState := #statFBState; // Set error state number for diagnostic 
                                 #statErrorAutoCleared := TRUE;
                                 #statMqttCommandState := #MQTT_COMMAND_STATE_NO_PROCESSING;
                             END_CASE;

                             //When QOS = 2 and Pub Complete Receieved:
                             CASE #tempMqttPubCompRcv OF
                               #NO_RESPONSE:  // Idle
                                 ;
                               #RESPONSE_GOOD:  //When QOS = 2 and Pub Complete Receieved:
                                 //disable watchdog
                                 #statEnableTimerCommandWatchdog := FALSE;
                                 //Encoding done all sent
                                 #statPaketHeaderEncodeDone := FALSE;
                                 //Publish QoS 2 = Done
                                 #statDone := TRUE;
                                 #statMqttCommandState := #MQTT_COMMAND_STATE_NO_PROCESSING;
                                 // Set Status back to connected
                                 #statStatus := #STATUS_JOB_EXECUTED;
                               #RESPONSE_PAKET_ID_INVALID:
                                 #statStatus := #ERR_MQTT_PAKET_ID_INVALID; // Set correct status that identifies error clearly
                                 #statSubfunctionStatus := #ERR_MQTT_PAKET_ID_INVALID; // Status or return value of called FBs, FCs and system blocks
                                 #statFBErrorState := #statFBState; // Set error state number for diagnostic 
                                 #statErrorAutoCleared := TRUE;
                                 #statMqttCommandState := #MQTT_COMMAND_STATE_NO_PROCESSING;
                             END_CASE;
                           END_REGION MQTT_COMMAND_SEND_PUBLISH

                         #MQTT_COMMAND_STATE_BUILD_SUBSCRIBE:  // Statement section case 2 
                           REGION SUBSCRIBE_TO_TOPIC
                             //Remaining Length is the length of the variable header (PacketID, 2Bytes) plus the length of the Payload. 
                             //Max Len of Mqtt pakets is per Standard 268,435,455 Bytes (ff,ff,ff,7f)
                             //Calculate Remain Len will be
                             //Len of TOPIC   (max 3*16382 WChars= 49.146 Bytes)
                             //LenInfo Topic (2Byte)
                             //QoS of Topic (1Byte)
                             //
                             //Set Status
                             #statStatus := #STATUS_MQTT_SUBSCRIBE;
                             // Must obey, if not currently sending PubAck Msg on a subscription
                             // Else, try in the next cycle
                             IF #tempTsendcBusy = FALSE // when tsendC is ready
                               AND #tempTsendcDone = FALSE // tsendC did not finish in this cycle
                               AND #statTsendcReq = FALSE // TsendC request was not already requested by pub ack msg
                             THEN
                               IF #statPaketHeaderEncodeDone = FALSE THEN

                                 //Init
                                 #statSendPaketTotalRemLen := 0;
                                 #statSendBufferPos := 0;
                                 #statSubscribeQos := #qos;
                                 #statSubscribeTopicEncodeState := #FIRST_ENCODING;
                                 #statSubscribeTopicPos := #FIRST_CHARACTER;
                                 #statSubscribeTopicLenUtf8Encoded := 0;
                                 #statPaketId += 1;//increment
                                 #statSubscribeQosEncoded := FALSE;

                                 //check necessary boundaries

                                 IF LEN(#mqttTopic) = #LEN_NULL THEN
                                   #statStatus := #ERR_MQTT_COMMAND_SUBSCRIBE_TOPIC_INVALID; // Set correct status that identifies error clearly
                                   #statSubfunctionStatus := #ERR_MQTT_COMMAND_SUBSCRIBE_TOPIC_INVALID; // Status or return value of called FBs, FCs and system blocks
                                   #statFBErrorState := #statFBState; // Set error state number for diagnostic 
                                   #statErrorAutoCleared := TRUE;
                                   #statMqttCommandState := #MQTT_COMMAND_STATE_NO_PROCESSING;
                                 ELSIF #statSubscribeQos > #MQTT_QOS_1 THEN
                                   #statStatus := #ERR_QOS_INVALID; // Set correct status that identifies error clearly
                                   #statSubfunctionStatus := #ERR_QOS_INVALID; // Status or return value of called FBs, FCs and system blocks
                                   #statFBErrorState := #statFBState; // Set error state number for diagnostic 
                                   #statErrorAutoCleared := TRUE;
                                   #statMqttCommandState := #MQTT_COMMAND_STATE_NO_PROCESSING;
                                 ELSE // All ok
                                   //Add two Byte for Paket ID:
                                   #statSendPaketTotalRemLen := #statSendPaketTotalRemLen + #TWO_BYTE_LEN_INFO;
                                   //Add one Byte for QoS Info:
                                   #statSendPaketTotalRemLen := #statSendPaketTotalRemLen + #ONE_BYTE_LEN_INFO;
                                   //add subscribe  topic len
                                   FOR #tempLoopCounter := #FIRST_CHARACTER TO LEN(#mqttTopic) DO
                                     "LMQTT_ConvertToUtf8"(character     := #mqttTopic[#tempLoopCounter],
                                                           convertedUtf8 => #tempConvertedUtf8,
                                                           bytesUsed     => #tempBytesUsedUtf8,
                                                           error         => #tempErrorConvertUtf8,
                                                           status        => #tempStatusConvertUtf8);
                                     #statSubscribeTopicLenUtf8Encoded := #statSubscribeTopicLenUtf8Encoded + #tempBytesUsedUtf8;
                                   END_FOR;
                                   //Add len of topic plus len info
                                   #statSendPaketTotalRemLen := #statSendPaketTotalRemLen + #statSubscribeTopicLenUtf8Encoded + #TWO_BYTE_LEN_INFO;

                                   //Build Subscribe Telegram
                                   //Fixed Header - Write Paket Type
                                   #statSendBuffer[#statSendBufferPos] := #MQTT_MSG_TYPE_SUBSCRIBE;
                                   #statSendBufferPos += 1; // increment

                                   //Write Remaining Paket Len info 
                                   WHILE (#statSendPaketTotalRemLen > #DEFAULT_VALUE_ZERO)
                                   DO//See MQTT Spec for explanation of this calculation
                                     #statEncodedRemPaketLenAsByte := UDINT_TO_BYTE(#statSendPaketTotalRemLen MOD #SEND_LEN_MULTIPLIER_UDINT_128);
                                     #statSendPaketTotalRemLen := #statSendPaketTotalRemLen / #SEND_LEN_MULTIPLIER_UDINT_128;
                                     // if there are more data to encode, set the top bit of this byte
                                     IF #statSendPaketTotalRemLen > #DEFAULT_VALUE_ZERO
                                     THEN
                                       // Do this and continue while loop
                                       #statEncodedRemPaketLenAsByte := #statEncodedRemPaketLenAsByte OR UDINT_TO_BYTE(#SEND_LEN_MULTIPLIER_UDINT_128);
                                       #statSendBuffer[#statSendBufferPos] := #statEncodedRemPaketLenAsByte;
                                       #statSendBufferPos += 1;
                                     ELSE
                                       //do this and leave while loop
                                       #statSendBuffer[#statSendBufferPos] := #statEncodedRemPaketLenAsByte;
                                       #statSendBufferPos += 1;
                                     END_IF;
                                   END_WHILE;

                                   // Set Paket Id
                                   #tempWordForSliceAddress := UINT_TO_WORD(#statPaketId);
                                   #statSendBuffer[#statSendBufferPos] := #tempWordForSliceAddress.%B1; //MSB
                                   #statSendBufferPos += 1;
                                   #statSendBuffer[#statSendBufferPos] := #tempWordForSliceAddress.%B0; //LSB
                                   #statSendBufferPos += 1;

                                   //When all done, set encode to true
                                   #statPaketHeaderEncodeDone := TRUE;
                                 END_IF;
                               END_IF;
                               //Header Encoded 
                               IF #statPaketHeaderEncodeDone = TRUE THEN
                                 //Header Encoded - now Topic and qos encoding

                                 //Subscribe Topic
                                 IF #statSendBufferPos <= #MAX_BUFFER_LEN_SEND - #TWO_BYTE_LEN_INFO THEN
                                   CASE #statSubscribeTopicEncodeState OF
                                     #FIRST_ENCODING:  // Statement section case 1
                                       //ADD len info into paket

                                       #tempWordForSliceAddress := UINT_TO_WORD(#statSubscribeTopicLenUtf8Encoded);
                                       #statSendBuffer[#statSendBufferPos] := #tempWordForSliceAddress.%B1; //MSB
                                       #statSendBufferPos += 1;
                                       #statSendBuffer[#statSendBufferPos] := #tempWordForSliceAddress.%B0; // LSB
                                       #statSendBufferPos += 1;

                                       FOR #tempLoopCounter := #statSubscribeTopicPos TO LEN(#mqttTopic) DO
                                         "LMQTT_ConvertToUtf8"(character     := #mqttTopic[#tempLoopCounter],
                                                               convertedUtf8 => #tempConvertedUtf8,
                                                               bytesUsed     => #tempBytesUsedUtf8,
                                                               error         => #tempErrorConvertUtf8,
                                                               status        => #tempStatusConvertUtf8);

                                         IF #statSendBufferPos + #tempBytesUsedUtf8 <= #MAX_BUFFER_LEN_SEND THEN
                                           #statSubscribeTopicPos += 1;
                                           CASE #tempBytesUsedUtf8 OF
                                             #UTF_1_BYTE_USED:  // Statement section case 1
                                               #statSendBuffer[#statSendBufferPos] := #tempConvertedUtf8.%B0;
                                               #statSendBufferPos += 1;
                                             #UTF_2_BYTE_USED:
                                               #statSendBuffer[#statSendBufferPos] := #tempConvertedUtf8.%B0;
                                               #statSendBufferPos += 1;
                                               #statSendBuffer[#statSendBufferPos] := #tempConvertedUtf8.%B1;
                                               #statSendBufferPos += 1;
                                             #UTF_3_BYTE_USED:  // Statement section case 2 to 4
                                               #statSendBuffer[#statSendBufferPos] := #tempConvertedUtf8.%B0;
                                               #statSendBufferPos += 1;
                                               #statSendBuffer[#statSendBufferPos] := #tempConvertedUtf8.%B1;
                                               #statSendBufferPos += 1;
                                               #statSendBuffer[#statSendBufferPos] := #tempConvertedUtf8.%B2;
                                               #statSendBufferPos += 1;
                                             ELSE  // Statement section ELSE
                                               ;
                                           END_CASE;
                                         ELSE
                                           //When buffer full
                                           #statSubscribeTopicEncodeState := #SUBSEQUENT_ENCODING;
                                           EXIT;
                                         END_IF;
                                       END_FOR;
                                       IF #statSubscribeTopicPos >= LEN(#mqttTopic) THEN
                                         #statSubscribeTopicEncodeState := #ENCODE_DONE;
                                       END_IF;

                                     #SUBSEQUENT_ENCODING:  // Statement section case 2 to 4
                                       FOR #tempLoopCounter := #statSubscribeTopicPos TO LEN(#mqttTopic) DO

                                         "LMQTT_ConvertToUtf8"(character     := #mqttTopic[#tempLoopCounter],
                                                               convertedUtf8 => #tempConvertedUtf8,
                                                               bytesUsed     => #tempBytesUsedUtf8,
                                                               error         => #tempErrorConvertUtf8,
                                                               status        => #tempStatusConvertUtf8);
                                         IF #statSendBufferPos + #tempBytesUsedUtf8 <= #MAX_BUFFER_LEN_SEND THEN
                                           #statSubscribeTopicPos += 1;
                                           CASE #tempBytesUsedUtf8 OF
                                             #UTF_1_BYTE_USED:  // Statement section case 1
                                               #statSendBuffer[#statSendBufferPos] := #tempConvertedUtf8.%B0;
                                               #statSendBufferPos += 1;
                                             #UTF_2_BYTE_USED:
                                               #statSendBuffer[#statSendBufferPos] := #tempConvertedUtf8.%B0;
                                               #statSendBufferPos += 1;
                                               #statSendBuffer[#statSendBufferPos] := #tempConvertedUtf8.%B1;
                                               #statSendBufferPos += 1;
                                             #UTF_3_BYTE_USED:  // Statement section case 2 to 4
                                               #statSendBuffer[#statSendBufferPos] := #tempConvertedUtf8.%B0;
                                               #statSendBufferPos += 1;
                                               #statSendBuffer[#statSendBufferPos] := #tempConvertedUtf8.%B1;
                                               #statSendBufferPos += 1;
                                               #statSendBuffer[#statSendBufferPos] := #tempConvertedUtf8.%B2;
                                               #statSendBufferPos += 1;
                                             ELSE  // Statement section ELSE
                                               ;
                                           END_CASE;
                                         ELSE
                                           //When buffer full
                                           EXIT;
                                         END_IF;
                                       END_FOR;
                                       IF #statSubscribeTopicPos >= LEN(#mqttTopic) THEN
                                         #statSubscribeTopicEncodeState := #ENCODE_DONE;
                                       END_IF;
                                     ELSE  // Skip when Done
                                       ;
                                   END_CASE;
                                 END_IF;

                                 IF #statSubscribeTopicEncodeState = #ENCODE_DONE
                                   AND #statSendBufferPos <= #MAX_BUFFER_LEN_SEND - #ONE_BYTE_LEN_INFO THEN
                                   #statSendBuffer[#statSendBufferPos] := USINT_TO_BYTE(#statSubscribeQos);
                                   #statSendBufferPos += 1;
                                   #statSubscribeQosEncoded := TRUE;
                                 END_IF;


                                 //set Sendlen for TSendC Block
                                 #statTsendcLen := #statSendBufferPos; // Buffer pos equals amount of elements in send array
                                 //reset buffer pos
                                 #statSendBufferPos := 0;
                                 //enable Send Req
                                 #statTsendcReq := TRUE;
                                 //Set Watchdog
                                 #statEnableTimerCommandWatchdog := TRUE;
                                 //wait for send to be done
                                 #statMqttCommandState := #MQTT_COMMAND_STATE_SEND_SUBSCRIBE;
                               END_IF;
                             END_IF;

                           END_REGION SUBSCRIBE_TO_TOPIC
                         #MQTT_COMMAND_STATE_SEND_SUBSCRIBE:
                           REGION SEND_SUBSCRIBE_WAIT_FOR_RESPONSE
                             //check tsend status
                             IF NOT #tempTsendcBusy AND #tempTsendcStatus = #TSENDC_JOB_DONE THEN
                               IF #statSubscribeTopicEncodeState = #ENCODE_DONE
                                 AND #statSubscribeQosEncoded = TRUE THEN
                                 //Encoding done all sent
                                 #statPaketHeaderEncodeDone := FALSE;
                               ELSE
                                 // More to Encode and send 
                                 #statEnableTimerCommandWatchdog := FALSE; // reset watchdog
                                 #statMqttCommandState := #MQTT_COMMAND_STATE_BUILD_SUBSCRIBE;
                               END_IF;
                             END_IF;
                             //Wait for timeout
                             IF #instTimerCommandWatchdog.Q THEN
                               #statEnableTimerCommandWatchdog := FALSE;
                               #statStatus := #ERR_MQTT_COMMAND_SEND_TIMEOUT; // Set correct status that identifies error clearly
                               #statSubfunctionStatus := #ERR_MQTT_COMMAND_SEND_TIMEOUT; // Status or return value of called FBs, FCs and system blocks
                               #statFBErrorState := #statFBState; // Set error state number for diagnostic 
                               #statErrorAutoCleared := TRUE;
                               #statMqttCommandState := #MQTT_COMMAND_STATE_NO_PROCESSING;
                             END_IF;

                             //Check Subscribe ACK paket
                             CASE #tempMqttSubAckRcv OF
                               #NO_RESPONSE:  // Statement section case 1
                                 ;
                               #RESPONSE_GOOD:  // Statement section case 2 to 4
                                 //disable watchdog
                                 #statEnableTimerCommandWatchdog := FALSE;
                                 //Encoding done all sent
                                 #statPaketHeaderEncodeDone := FALSE;
                                 // Job done
                                 #statDone := TRUE;
                                 #statMqttCommandState := #MQTT_COMMAND_STATE_NO_PROCESSING;
                                 // Set Status back to connected
                                 #statStatus := #STATUS_JOB_EXECUTED;
                               #RESPONSE_PAKET_ID_INVALID:  // PaketId Invalid
                                 #statStatus := #ERR_MQTT_PAKET_ID_INVALID; // Set correct status that identifies error clearly
                                 #statSubfunctionStatus := #ERR_MQTT_PAKET_ID_INVALID; // Status or return value of called FBs, FCs and system blocks
                                 #statFBErrorState := #statFBState; // Set error state number for diagnostic 
                                 #statErrorAutoCleared := TRUE;
                                 #statMqttCommandState := #MQTT_COMMAND_STATE_NO_PROCESSING;
                               #RESPONSE_SUBSCRIBE_FAILED:
                                 #statStatus := #ERR_MQTT_SUBACK_FAILURE; // Set correct status that identifies error clearly
                                 #statSubfunctionStatus := #ERR_MQTT_SUBACK_FAILURE; // Status or return value of called FBs, FCs and system blocks
                                 #statFBErrorState := #statFBState; // Set error state number for diagnostic 
                                 #statErrorAutoCleared := TRUE;
                                 #statMqttCommandState := #MQTT_COMMAND_STATE_NO_PROCESSING;
                             END_CASE;
                           END_REGION SEND_SUBSCRIBE_WAIT_FOR_RESPONSE

                         #MQTT_COMMAND_STATE_BUILD_UNSUBSCRIBE:// Unsubscribe from topics
                           REGION UNSUBSCRIBE_FROM_TOPIC
                             //Remaining Length is the length of the variable header (PacketID, 2Bytes) plus the length of the Payload. 
                             //Max Len of Mqtt pakets is per Standard 268,435,455 Bytes (ff,ff,ff,7f)
                             //Calculate Remain Len will be
                             //Len of TOPIC   (max 3*16382 WChars= 49.146 Bytes)
                             //LenInfo Topic (2Byte)
                             //
                             //Set Status
                             #statStatus := #STATUS_MQTT_UNSUBSCRIBE;
                             // Must obey, if not currently sending PubAck Msg on a subscription
                             // Else, try in the next cycle
                             IF #tempTsendcBusy = FALSE // when tsendC is ready
                               AND #tempTsendcDone = FALSE // tsendC did not finish in this cycle
                               AND #statTsendcReq = FALSE // TsendC request was not already requested by pub ack msg
                             THEN
                               //Header not encoded
                               IF #statPaketHeaderEncodeDone = FALSE THEN
                                 //Init
                                 #statSendPaketTotalRemLen := 0;
                                 #statSendBufferPos := 0;
                                 #statUnsubscribeTopicEncodeState := #FIRST_ENCODING;
                                 #statUnsubscribeTopicPos := #FIRST_CHARACTER;
                                 #statUnsubscribeTopicLenUtf8Encoded := 0;
                                 #statPaketId += 1;//increment

                                 //check necessary boundaries

                                 IF LEN(#mqttTopic) = #LEN_NULL THEN
                                   #statStatus := #ERR_MQTT_COMMAND_UNSUBSCRIBE_TOPIC_INVALID; // Set correct status that identifies error clearly
                                   #statSubfunctionStatus := #ERR_MQTT_COMMAND_UNSUBSCRIBE_TOPIC_INVALID; // Status or return value of called FBs, FCs and system blocks
                                   #statFBErrorState := #statFBState; // Set error state number for diagnostic 
                                   #statErrorUserCleared := TRUE;
                                 ELSE // All ok
                                   //Add two Byte for Paket ID:
                                   #statSendPaketTotalRemLen := #statSendPaketTotalRemLen + #TWO_BYTE_LEN_INFO;
                                   //add unsubscribe  topic len
                                   FOR #tempLoopCounter := #FIRST_CHARACTER TO LEN(#mqttTopic) DO
                                     "LMQTT_ConvertToUtf8"(character     := #mqttTopic[#tempLoopCounter],
                                                           convertedUtf8 => #tempConvertedUtf8,
                                                           bytesUsed     => #tempBytesUsedUtf8,
                                                           error         => #tempErrorConvertUtf8,
                                                           status        => #tempStatusConvertUtf8);
                                     #statUnsubscribeTopicLenUtf8Encoded := #statUnsubscribeTopicLenUtf8Encoded + #tempBytesUsedUtf8;
                                   END_FOR;
                                   //Add len of topic plus len info
                                   #statSendPaketTotalRemLen := #statSendPaketTotalRemLen + #statUnsubscribeTopicLenUtf8Encoded + #TWO_BYTE_LEN_INFO;

                                   //Build Subscribe Telegram
                                   //Fixed Header - Write Paket Type
                                   #statSendBuffer[#statSendBufferPos] := #MQTT_MSG_TYPE_UNSUBSCRIBE;
                                   #statSendBufferPos += 1; // increment

                                   //Write Remaining Paket Len info 
                                   WHILE (#statSendPaketTotalRemLen > #DEFAULT_VALUE_ZERO)
                                   DO//See MQTT Spec for explanation of this calculation
                                     #statEncodedRemPaketLenAsByte := UDINT_TO_BYTE(#statSendPaketTotalRemLen MOD #SEND_LEN_MULTIPLIER_UDINT_128);
                                     #statSendPaketTotalRemLen := #statSendPaketTotalRemLen / #SEND_LEN_MULTIPLIER_UDINT_128;
                                     // if there are more data to encode, set the top bit of this byte
                                     IF #statSendPaketTotalRemLen > #DEFAULT_VALUE_ZERO
                                     THEN
                                       // Do this and continue while loop
                                       #statEncodedRemPaketLenAsByte := #statEncodedRemPaketLenAsByte OR UDINT_TO_BYTE(#SEND_LEN_MULTIPLIER_UDINT_128);
                                       #statSendBuffer[#statSendBufferPos] := #statEncodedRemPaketLenAsByte;
                                       #statSendBufferPos += 1;
                                     ELSE
                                       //do this and leave while loop
                                       #statSendBuffer[#statSendBufferPos] := #statEncodedRemPaketLenAsByte;
                                       #statSendBufferPos += 1;
                                     END_IF;
                                   END_WHILE;

                                   // Set Paket Id
                                   #tempWordForSliceAddress := UINT_TO_WORD(#statPaketId);
                                   #statSendBuffer[#statSendBufferPos] := #tempWordForSliceAddress.%B1; //MSB
                                   #statSendBufferPos += 1;
                                   #statSendBuffer[#statSendBufferPos] := #tempWordForSliceAddress.%B0; //LSB
                                   #statSendBufferPos += 1;

                                   //When all done, set encode to true
                                   #statPaketHeaderEncodeDone := TRUE;
                                 END_IF;
                               END_IF;

                               //Header Encoded - 
                               IF #statPaketHeaderEncodeDone = TRUE THEN
                                 //Unsubscribe Topic
                                 IF #statSendBufferPos <= #MAX_BUFFER_LEN_SEND - #TWO_BYTE_LEN_INFO THEN
                                   CASE #statUnsubscribeTopicEncodeState OF
                                     #FIRST_ENCODING:  // Statement section case 1
                                       //ADD len info into paket

                                       #tempWordForSliceAddress := UINT_TO_WORD(#statUnsubscribeTopicLenUtf8Encoded);
                                       #statSendBuffer[#statSendBufferPos] := #tempWordForSliceAddress.%B1; //MSB
                                       #statSendBufferPos += 1;
                                       #statSendBuffer[#statSendBufferPos] := #tempWordForSliceAddress.%B0; // LSB
                                       #statSendBufferPos += 1;

                                       FOR #tempLoopCounter := #statUnsubscribeTopicPos TO LEN(#mqttTopic) DO
                                         "LMQTT_ConvertToUtf8"(character     := #mqttTopic[#tempLoopCounter],
                                                               convertedUtf8 => #tempConvertedUtf8,
                                                               bytesUsed     => #tempBytesUsedUtf8,
                                                               error         => #tempErrorConvertUtf8,
                                                               status        => #tempStatusConvertUtf8);

